{attribute addProperty BoxType "IODEVICETYPE_ETHERCATPROT"}
{attribute addProperty Id "Beckhoff_BKxxxxBeckhoff_BKxxxx_655B233100Beckhoff_CUxxxxBeckhoff_CUxxxx_D794C9731008126Beckhoff_CXxxxxBeckhoff_CXxxxx_51161BB04544568TcTerminals210_EK1100_1TcTerminals210_EK1100_1_99191ECD00TcTerminals210_EK1100_2TcTerminals210_EK1100_2_BDAFA3B600SyncUnitsSyncUnits_3FA29F3C21627InputsInputs_C75D3FEC1280160OutputsOutputs_47D1E803848106InfoDataInfoData_45F98C5022428"}
{attribute addProperty CRC "1289812287"}
{attribute addProperty SizeInBites "8120"}
{attribute addProperty SizeInBytes "1015"}
TYPE EtherCAT_Master_BKCUCX_4CE0F93F :
STRUCT
	{attribute addProperty Name "Beckhoff_BKxxxx"}
	Beckhoff_BKxxxx : Beckhoff_BKxxxx_655B2331;
	{attribute addProperty Name "Beckhoff_CUxxxx"}
	Beckhoff_CUxxxx : Beckhoff_CUxxxx_D794C973;
	{attribute addProperty Name "Beckhoff_CXxxxx"}
	Beckhoff_CXxxxx : Beckhoff_CXxxxx_51161BB0;
	{attribute addProperty Name "TcTerminals210_EK1100_1"}
	TcTerminals210_EK1100_1 : TcTerminals210_EK1100_1_99191ECD;
	{attribute addProperty Name "TcTerminals210_EK1100_2"}
	TcTerminals210_EK1100_2 : TcTerminals210_EK1100_2_BDAFA3B6;
	{attribute addProperty Name "SyncUnits"}
	SyncUnits : SyncUnits_3FA29F3C;
	{attribute addProperty Name "Inputs"}
	Inputs : Inputs_C75D3FEC;
	{attribute addProperty Name "Outputs"}
	Outputs : Outputs_47D1E803;
	{attribute addProperty Name "InfoData"}
	InfoData : InfoData_45F98C50;
END_STRUCT
END_TYPE

(* stored: Version 1.2.0.0, ProductVersion 3.1.4024.9
   DUT EtherCAT_Master_BKCUCX_4CE0F93F: Id {027d7849-6123-42f4-a950-ff91b3208a6a} *)
